(* IEC 61131-3 sources: HvIrBz/, 6 files *)

(* ---- d512.st ---- *)
if 取出物料盒1=1 THEN
	X轴绝对运动启动:=0;
	Z轴绝对运动启动:=0;
	X轴绝对运动位置设定 := 572;
    Z轴绝对运动位置设定 := 280;
	x回原点:=0;
	y回原点:=0;
	z回原点:=0;
(*	xz轴设定终了:=1;*)
	Y0 :=1;
	y3 :=0;
	Y1 :=0;
	X轴绝对运动速度设定:=50;
	Z轴绝对运动速度设定:=50;
	X轴绝对运动启动:=1;
	Z轴绝对运动启动:=1;

END_IF

if Z轴实时位置=280 and X轴实时位置=572 then
		旋转气缸:=1;
		Y轴绝对运动位置设定:=-188;
		Y轴绝对运动速度设定:=50;
		Y轴绝对运动启动:=1;
		y3 :=1;
END_IF

if 取出物料盒2=1 THEN
	X轴绝对运动位置设定 := 432;
    Z轴绝对运动位置设定 := 280;
x回原点:=0;
	y回原点:=0;
	z回原点:=0;
(*	xz轴设定终了:=1;*)
	Y0 :=1;
	y3 :=0;
	Y1 :=0;
	X轴绝对运动速度设定:=50;
	Z轴绝对运动速度设定:=50;
	X轴绝对运动启动:=1;
	Z轴绝对运动启动:=1;

END_IF

if Z轴实时位置=280 and X轴实时位置=432 then
		旋转气缸:=1;
		Y轴绝对运动位置设定:=-188;
		Y轴绝对运动速度设定:=50;
		Y轴绝对运动启动:=1;
		y3 :=1;
END_IF

if 取出物料盒3=1 THEN
	X轴绝对运动位置设定 := 292;
    Z轴绝对运动位置设定 := 280;
x回原点:=0;
	y回原点:=0;
	z回原点:=0;
(*	xz轴设定终了:=1;*)
	Y0 :=1;
	y3 :=0;
	Y1 :=0;
	X轴绝对运动速度设定:=50;
	Z轴绝对运动速度设定:=50;
	X轴绝对运动启动:=1;
	Z轴绝对运动启动:=1;

END_IF

if Z轴实时位置=280 and X轴实时位置=292 then
		旋转气缸:=1;
		Y轴绝对运动位置设定:=-188;
		Y轴绝对运动速度设定:=50;
		Y轴绝对运动启动:=1;
		y3 :=1;
		Y轴绝对运动启动:=0;
END_IF

if 取出物料盒4=1 THEN
	X轴绝对运动位置设定 := 152;
    Z轴绝对运动位置设定 := 280;
x回原点:=0;
	y回原点:=0;
	z回原点:=0;
(*	xz轴设定终了:=1;*)
	Y0 :=1;
	y3 :=0;
	Y1 :=0;
	X轴绝对运动速度设定:=50;
	Z轴绝对运动速度设定:=50;
	X轴绝对运动启动:=1;
	Z轴绝对运动启动:=1;
	X轴绝对运动启动:=0;
	Z轴绝对运动启动:=0;

END_IF

if Z轴实时位置=280 and X轴实时位置=152  then
		旋转气缸:=1;
		Z轴绝对运动启动:=0;
		Y轴绝对运动位置设定:=-188;
		Y轴绝对运动速度设定:=50;
		Y轴绝对运动启动:=1;
		Z轴绝对运动启动:=0;
		Y轴绝对运动启动:=0;
		y3 :=1;
END_IF

if 取出物料盒5=1 THEN
	X轴绝对运动位置设定 := 12;
    Z轴绝对运动位置设定 := 280;
x回原点:=0;
	y回原点:=0;
	z回原点:=0;
(*	xz轴设定终了:=1;*)
	Y0 :=1;
	y3 :=0;
	Y1 :=0;
	X轴绝对运动速度设定:=50;
	Z轴绝对运动速度设定:=50;
	X轴绝对运动启动:=1;
	Z轴绝对运动启动:=1;
	X轴绝对运动启动:=0;
	Z轴绝对运动启动:=0;

END_IF

if Z轴实时位置=280 and X轴实时位置=12  then
		旋转气缸:=1;
		Z轴绝对运动启动:=0;
		Y轴绝对运动位置设定:=-188;
		Y轴绝对运动速度设定:=50;
		Y轴绝对运动启动:=1;
		Z轴绝对运动启动:=0;
		Y轴绝对运动启动:=0;
		y3 :=1;
END_IF

(*if 取出物料盒6=1 THEN
	X轴绝对运动启动:=0;
	Z轴绝对运动启动:=0;
	X轴绝对运动位置设定 := 572;
    Z轴绝对运动位置设定 := 135;
x回原点:=0;
	y回原点:=0;
	z回原点:=0;
(*	xz轴设定终了:=1;*)
	Y0 :=1;
	y3 :=0;
	Y1 :=0;
	X轴绝对运动速度设定:=50;
	Z轴绝对运动速度设定:=50;
	X轴绝对运动启动:=1;
	Z轴绝对运动启动:=1;

END_IF

if Z轴实时位置=135 and X轴实时位置=572 and y3=0 then
		旋转气缸:=1;
		Y轴绝对运动位置设定:=-188;
		Y轴绝对运动速度设定:=50;
		Y轴绝对运动启动:=1;
		y3 :=1;
END_IF

if 取出物料盒7=1 THEN
	X轴绝对运动位置设定 := 432;
    Z轴绝对运动位置设定 := 135;
x回原点:=0;
	y回原点:=0;
	z回原点:=0;
(*	xz轴设定终了:=1;*)
	Y0 :=1;
	y3 :=0;
	Y1 :=0;
	X轴绝对运动速度设定:=50;
	Z轴绝对运动速度设定:=50;
	X轴绝对运动启动:=1;
	Z轴绝对运动启动:=1;

END_IF

if Z轴实时位置=135 and X轴实时位置=432 then
		旋转气缸:=1;
		Y轴绝对运动位置设定:=-188;
		Y轴绝对运动速度设定:=50;
		Y轴绝对运动启动:=1;
		y3 :=1;
END_IF

if 取出物料盒8=1 THEN
	X轴绝对运动位置设定 := 292;
    Z轴绝对运动位置设定 := 135;
x回原点:=0;
	y回原点:=0;
	z回原点:=0;
(*	xz轴设定终了:=1;*)
	Y0 :=1;
	y3 :=0;
	Y1 :=0;
	X轴绝对运动速度设定:=50;
	Z轴绝对运动速度设定:=50;
	X轴绝对运动启动:=1;
	Z轴绝对运动启动:=1;

END_IF

if Z轴实时位置=135 and X轴实时位置=292 then
		旋转气缸:=1;
		Y轴绝对运动位置设定:=-188;
		Y轴绝对运动速度设定:=50;
		Y轴绝对运动启动:=1;
		y3 :=1;
		Y轴绝对运动启动:=0;
END_IF

if 取出物料盒9=1 THEN
	X轴绝对运动位置设定 := 152;
    Z轴绝对运动位置设定 := 135;
x回原点:=0;
	y回原点:=0;
	z回原点:=0;
(*	xz轴设定终了:=1;*)
	Y0 :=1;
	y3 :=0;
	Y1 :=0;
	X轴绝对运动速度设定:=50;
	Z轴绝对运动速度设定:=50;
	X轴绝对运动启动:=1;
	Z轴绝对运动启动:=1;
	X轴绝对运动启动:=0;
	Z轴绝对运动启动:=0;

END_IF

if Z轴实时位置=135 and X轴实时位置=152 and 旋转气缸=0 then
		旋转气缸:=1;
		Z轴绝对运动启动:=0;
		Y轴绝对运动位置设定:=-188;
		Y轴绝对运动速度设定:=50;
		Y轴绝对运动启动:=1;
		Z轴绝对运动启动:=0;
		Y轴绝对运动启动:=0;
		y3 :=1;
END_IF

if 取出物料盒10=1 THEN
	X轴绝对运动位置设定 := 12;
    Z轴绝对运动位置设定 := 135;
x回原点:=0;
	y回原点:=0;
	z回原点:=0;
(*	xz轴设定终了:=1;*)
	Y0 :=1;
	y3 :=0;
	Y1 :=0;
	X轴绝对运动速度设定:=50;
	Z轴绝对运动速度设定:=50;
	X轴绝对运动启动:=1;
	Z轴绝对运动启动:=1;
	X轴绝对运动启动:=0;
	Z轴绝对运动启动:=0;

END_IF

if Z轴实时位置=135 and X轴实时位置=12 and 旋转气缸=0 then
		旋转气缸:=1;
		Z轴绝对运动启动:=0;
		Y轴绝对运动位置设定:=-188;
		Y轴绝对运动速度设定:=50;
		Y轴绝对运动启动:=1;
		Z轴绝对运动启动:=0;
		Y轴绝对运动启动:=0;
		y3 :=1;
END_IF

if 取出物料盒11=1 THEN
	X轴绝对运动启动:=0;
	Z轴绝对运动启动:=0;
	X轴绝对运动位置设定 := 572;
    Z轴绝对运动位置设定 := -10;
x回原点:=0;
	y回原点:=0;
	z回原点:=0;
(*	xz轴设定终了:=1;*)
	Y0 :=1;
	y3 :=0;
	Y1 :=0;
	X轴绝对运动速度设定:=50;
	Z轴绝对运动速度设定:=50;
	X轴绝对运动启动:=1;
	Z轴绝对运动启动:=1;

END_IF

if Z轴实时位置=-10 and X轴实时位置=572 and y3=0 then
		旋转气缸:=1;
		Y轴绝对运动位置设定:=-188;
		Y轴绝对运动速度设定:=50;
		Y轴绝对运动启动:=1;
		y3 :=1;
END_IF

if 取出物料盒12=1 THEN
	X轴绝对运动位置设定 := 432;
    Z轴绝对运动位置设定 := -10;
x回原点:=0;
	y回原点:=0;
	z回原点:=0;
(*	xz轴设定终了:=1;*)
	Y0 :=1;
	y3 :=0;
	Y1 :=0;
	X轴绝对运动速度设定:=50;
	Z轴绝对运动速度设定:=50;
	X轴绝对运动启动:=1;
	Z轴绝对运动启动:=1;

END_IF

if Z轴实时位置=-10 and X轴实时位置=432 then
		旋转气缸:=1;
		Y轴绝对运动位置设定:=-188;
		Y轴绝对运动速度设定:=50;
		Y轴绝对运动启动:=1;
		y3 :=1;
END_IF

if 取出物料盒13=1 THEN
	X轴绝对运动位置设定 := 292;
    Z轴绝对运动位置设定 := -10;
x回原点:=0;
	y回原点:=0;
	z回原点:=0;
(*	xz轴设定终了:=1;*)
	Y0 :=1;
	y3 :=0;
	Y1 :=0;
	X轴绝对运动速度设定:=50;
	Z轴绝对运动速度设定:=50;
	X轴绝对运动启动:=1;
	Z轴绝对运动启动:=1;

END_IF

if Z轴实时位置=-10 and X轴实时位置=292 then
		旋转气缸:=1;
		Y轴绝对运动位置设定:=-188;
		Y轴绝对运动速度设定:=50;
		Y轴绝对运动启动:=1;
		y3 :=1;
		Y轴绝对运动启动:=0;
END_IF

if 取出物料盒14=1 THEN
	X轴绝对运动位置设定 := 152;
    Z轴绝对运动位置设定 := -10;
x回原点:=0;
	y回原点:=0;
	z回原点:=0;
(*	xz轴设定终了:=1;*)
	Y0 :=1;
	y3 :=0;
	Y1 :=0;
	X轴绝对运动速度设定:=50;
	Z轴绝对运动速度设定:=50;
	X轴绝对运动启动:=1;
	Z轴绝对运动启动:=1;
	X轴绝对运动启动:=0;
	Z轴绝对运动启动:=0;

END_IF

if Z轴实时位置=-10 and X轴实时位置=152 and 旋转气缸=0 then
		旋转气缸:=1;
		Z轴绝对运动启动:=0;
		Y轴绝对运动位置设定:=-188;
		Y轴绝对运动速度设定:=50;
		Y轴绝对运动启动:=1;
		Z轴绝对运动启动:=0;
		Y轴绝对运动启动:=0;
		y3 :=1;
END_IF

if 取出物料盒15=1 THEN
	X轴绝对运动位置设定 := 12;
    Z轴绝对运动位置设定 := -10;
x回原点:=0;
	y回原点:=0;
	z回原点:=0;
(*	xz轴设定终了:=1;*)
	Y0 :=1;
	y3 :=0;
	Y1 :=0;
	X轴绝对运动速度设定:=50;
	Z轴绝对运动速度设定:=50;
	X轴绝对运动启动:=1;
	Z轴绝对运动启动:=1;
	X轴绝对运动启动:=0;
	Z轴绝对运动启动:=0;

END_IF

if Z轴实时位置=-10 and X轴实时位置=12 and 旋转气缸=0 then
		旋转气缸:=1;
		Z轴绝对运动启动:=0;
		Y轴绝对运动位置设定:=-188;
		Y轴绝对运动速度设定:=50;
		Y轴绝对运动启动:=1;
		Z轴绝对运动启动:=0;
		Y轴绝对运动启动:=0;
		y3 :=1;
END_IF*)

if x5=1 THEN
	Z轴绝对运动启动:=0;
	Y轴绝对运动启动:=0;
	END_IF

if Y轴实时位置=-188 then
	Z轴绝对运动启动:=0;
	Y轴绝对运动启动:=0;
	夹爪气缸:=1;
	y3:=0;
	Y2:=1;
	Z轴绝对运动位置设定:=285;
	Y轴绝对运动位置设定:=40;
	Z轴绝对运动速度设定:=50;
	Y轴绝对运动速度设定:=50;
(*	Z轴绝对运动启动:=1;
	Y轴绝对运动启动:=1;*)

	END_IF

if x6=1 THEN

	Z轴绝对运动启动:=1;
	Y轴绝对运动启动:=1;

	END_IF
(*if 取出物料盒2=1 or X6=1 THEN
	X轴绝对运动位置设定 := 432;
    Z轴绝对运动位置设定 := 280;

	xz轴设定终了:=1;
	Y1 :=1;
	Y0 :=0;
(*	X轴绝对运动启动:=1;
	Z轴绝对运动启动:=1;*)
END_IF

if 取出物料盒3=1 THEN
	X轴绝对运动位置设定 := 292;
    Z轴绝对运动位置设定 := 280;

	xz轴设定终了:=1;
	Y1 :=1;
	Y0 :=0;
(*	X轴绝对运动启动:=1;
	Z轴绝对运动启动:=1;*)
END_IF

if 取出物料盒4=1 THEN
	X轴绝对运动位置设定 := 152;
    Z轴绝对运动位置设定 := 280;

	xz轴设定终了:=1;
	Y1 :=1;
	Y0 :=0;
(*	X轴绝对运动启动:=1;
	Z轴绝对运动启动:=1;*)
END_IF

(*if 取出物料盒5=1 THEN
	X轴绝对运动位置设定 := 12;
    Z轴绝对运动位置设定 := 280;

	xz轴设定终了:=1;
	Y1 :=1;
	Y0 :=0;
	X轴绝对运动启动:=1;
	Z轴绝对运动启动:=1;
END_IF*)

if 取出物料盒1=1 or X6=1 THEN
	X轴绝对运动位置设定 := 432;
    Z轴绝对运动位置设定 := 280;

	xz轴设定终了:=1;
	Y1 :=1;
	Y0 :=0;
	X轴绝对运动启动:=1;
	Z轴绝对运动启动:=1;
END_IF

IF X5=1 THEN
	x回原点:=0;
	y回原点:=0;
	z回原点:=0;
	旋转气缸:=1;
	Y轴绝对运动位置设定:=-188;
	Y轴绝对运动速度设定:=50;
	X轴绝对运动速度设定:=50;
	Z轴绝对运动速度设定:=50;
	Y轴绝对运动启动:=1;
	X轴绝对运动启动:=1;
	Z轴绝对运动启动:=1;
	夹爪气缸:=1;
	IF Y轴实时位置=-188 THEN
	Y3:=1;
	END_IF;
END_IF*)

if X4=1 THEN
	旋转气缸:=0;
	x回原点:=1;
	y回原点:=1;
	z回原点:=1;
	X轴绝对运动启动:=0;
	Y轴绝对运动启动:=0;
	Z轴绝对运动启动:=0;
	END_IF

(* ---- d514.st ---- *)
if M8000=1 and 初始启动一次=0 THEN
	Z轴绝对运动启动:=0;
	X轴绝对运动启动:=0;
	Y轴绝对运动启动:=0;
	x回原点:=0;
	y回原点:=0;
	z回原点:=0;
	X轴绝对运动速度设定:=50;
	Z轴绝对运动速度设定:=50;
	y1:=1;
	d1301:=0;
	三轴启动:=0;
	初始启动一次:=1;
END_IF

IF 三轴启动=1 THEN
	X轴绝对运动速度设定:=50;
	Z轴绝对运动速度设定:=50;
	CASE 第一个运行 OF
		1:取出物料盒1:=1;
		2:取出物料盒2:=1;
		3:取出物料盒3:=1;
		4:取出物料盒4:=1;
		5:取出物料盒5:=1;
	Z轴绝对运动启动:=0;
	X轴绝对运动启动:=0;
	END_CASE;
END_IF;
if 取出物料盒1=1 and 取出物料盒只执行一次确保=0 THEN
	取出1:=1;
	X轴绝对运动位置设定 := 572;
    Z轴绝对运动位置设定 := 280;
	Z轴绝对运动启动:=1;
	取得是1:=1;
	取出物料盒只执行一次确保:=1;
END_IF
if 取出物料盒2=1 THEN
	取出1:=1;
	X轴绝对运动位置设定 := 432;
    Z轴绝对运动位置设定 := 280;
	Z轴绝对运动启动:=1;
	取得是2:=1;

END_IF
if  取出物料盒3=1  THEN
	取出1:=1;
	X轴绝对运动位置设定 := 292;
    Z轴绝对运动位置设定 := 280;
	Z轴绝对运动启动:=1;
	取得是3:=1;
END_IF
if 取出物料盒4=1 THEN
	取出1:=1;
	X轴绝对运动位置设定 := 152;
    Z轴绝对运动位置设定 := 280;
	Z轴绝对运动启动:=1;
	取得是4:=1;
END_IF
if  取出物料盒5=1 THEN
	取出1:=1;
	X轴绝对运动位置设定 := 12;
    Z轴绝对运动位置设定 := 280;
	Z轴绝对运动启动:=1;
	取得是5:=1;
END_IF
	IF Z轴实时位置>20 and 取得是1=1  THEN

		X轴绝对运动启动:=1;
	END_IF;

	IF Z轴实时位置>20 and 取得是2=1  THEN

		X轴绝对运动启动:=1;
	END_IF;

	IF Z轴实时位置>20 and 取得是3=1  THEN

		X轴绝对运动启动:=1;
	END_IF;

	IF Z轴实时位置>20 and 取得是4=1  THEN

		X轴绝对运动启动:=1;
	END_IF;

	IF Z轴实时位置>20 and 取得是5=1  THEN

		X轴绝对运动启动:=1;
	END_IF;
if Z轴实时位置=280 and X轴实时位置=572 and 取得是1=1 then
		旋转气缸:=1;
		Y轴绝对运动位置设定:=-188;
		Y轴绝对运动速度设定:=50;
		Y轴绝对运动启动:=1;
		y3 :=1;
		Z轴绝对运动启动:=0;
END_IF

if Z轴实时位置=280 and X轴实时位置=432 and 取得是2=1 then
		旋转气缸:=1;
		Y轴绝对运动位置设定:=-188;
		Y轴绝对运动速度设定:=50;
		Y轴绝对运动启动:=1;
		y3 :=1;
END_IF

if Z轴实时位置=280 and X轴实时位置=292 and 取得是3=1 then
		旋转气缸:=1;
		Y轴绝对运动位置设定:=-188;
		Y轴绝对运动速度设定:=50;
		Y轴绝对运动启动:=1;
		y3 :=1;
END_IF

if Z轴实时位置=280 and X轴实时位置=152 and 取得是4=1 then
		旋转气缸:=1;
		Y轴绝对运动位置设定:=-188;
		Y轴绝对运动速度设定:=50;
		Y轴绝对运动启动:=1;
		y3 :=1;
END_IF
if Z轴实时位置=280 and X轴实时位置=12 and 取得是5=1 then
		旋转气缸:=1;
		Y轴绝对运动位置设定:=-188;
		Y轴绝对运动速度设定:=50;
		Y轴绝对运动启动:=1;
		y3 :=1;
END_IF
if Y轴实时位置=-188 then
	Z轴绝对运动启动:=0;
	Y轴绝对运动启动:=0;
	夹爪气缸:=1;
	y3:=0;
	Y2:=1;
	Z轴绝对运动位置设定:=285;
	Y轴绝对运动位置设定:=40;
	Z轴绝对运动速度设定:=50;
	Y轴绝对运动速度设定:=50;
	X轴绝对运动位置设定:=303;
	Z轴绝对运动启动:=1;
	END_IF

IF Z轴实时位置=285 THEN

	Y轴绝对运动启动:=1;
	运动状态:=0;
	取料终:=1;
END_IF;

(*IF x5=1 THEN
	Z轴绝对运动启动:=1;
	Y轴绝对运动启动:=1;
	运动状态:=0;
	取料终:=1;
END_IF;*)

IF 取料终=1 and Y轴实时位置>35 THEN
	旋转气缸:=0;
	X轴绝对运动启动:=1;
	放到顶上了:=1;
	Z轴绝对运动启动:=0;
	Y轴绝对运动启动:=0;
	Y2:=1;
END_IF;

IF 放到顶上了=1 and X轴实时位置=303 THEN
	Z轴绝对运动位置设定:=0;
	Z轴绝对运动启动:=1;
	Y轴绝对运动启动:=1;
	X轴绝对运动启动:=1;
	Y3:=1;
	放完了:=1;
END_IF;

IF 放完了=1 and Z轴实时位置=0 THEN
	夹爪气缸:=0;
	x回原点:=1;
	y回原点:=1;
	z回原点:=1;
END_IF;

(* ---- d515.st ---- *)
if M8000=1 and 初始启动一次=0 THEN
	Z轴绝对运动启动:=0;
	X轴绝对运动启动:=0;
	Y轴绝对运动启动:=0;
	x回原点:=0;
	y回原点:=0;
	z回原点:=0;
	X轴绝对运动速度设定:=50;
	Z轴绝对运动速度设定:=50;

	d1301:=0;
	三轴启动:=0;
	圆形落料:=0;
	初始启动一次:=1;

END_IF

IF 三轴启动=1 THEN
	传送带速度:=50;
	传送带位置:=20000;
	圆形物料推料气缸:=1;

	切换吸盘:=1;

	X轴绝对运动速度设定:=50;
	Z轴绝对运动速度设定:=50;
	CASE 第一个运行 OF
		1:取出物料盒1:=1;
		2:取出物料盒2:=1;
		3:取出物料盒3:=1;
		4:取出物料盒4:=1;
		5:取出物料盒5:=1;
		6:取出物料盒6:=1;
		7:取出物料盒7:=1;
		8:取出物料盒8:=1;
		9:取出物料盒9:=1;
		10:取出物料盒10:=1;
		11:取出物料盒11:=1;
		12:取出物料盒12:=1;
		13:取出物料盒13:=1;
		14:取出物料盒14:=1;
		15:取出物料盒15:=1;

	Z轴绝对运动启动:=0;
	X轴绝对运动启动:=0;
	END_CASE;
END_IF;
if 取出物料盒1=1 and 取出物料盒只执行一次确保=0 THEN
	取出1:=1;
	X轴绝对运动位置设定 := 572;
    Z轴绝对运动位置设定 := 280;
	Z轴绝对运动启动:=1;
	取得是1:=1;
	取出物料盒只执行一次确保:=1;
END_IF
if 取出物料盒2=1 and 取出物料盒只执行一次确保=0 THEN
	取出1:=1;
	X轴绝对运动位置设定 := 432;
    Z轴绝对运动位置设定 := 280;
	Z轴绝对运动启动:=1;
	取得是2:=1;
	取出物料盒只执行一次确保:=1;
END_IF
if  取出物料盒3=1 and 取出物料盒只执行一次确保=0  THEN
	取出1:=1;
	X轴绝对运动位置设定 := 292;
    Z轴绝对运动位置设定 := 280;
	Z轴绝对运动启动:=1;
	取得是3:=1;
	取出物料盒只执行一次确保:=1;
END_IF
if 取出物料盒4=1 and 取出物料盒只执行一次确保=0 THEN
	取出1:=1;
	X轴绝对运动位置设定 := 152;
    Z轴绝对运动位置设定 := 280;
	Z轴绝对运动启动:=1;
	取得是4:=1;
	取出物料盒只执行一次确保:=1;
END_IF
if  取出物料盒5=1 and 取出物料盒只执行一次确保=0 THEN
	取出1:=1;
	X轴绝对运动位置设定 := 12;
    Z轴绝对运动位置设定 := 280;
	Z轴绝对运动启动:=1;
	取得是5:=1;
	取出物料盒只执行一次确保:=1;
END_IF
if 取出物料盒6=1 and 取出物料盒只执行一次确保=0 THEN
	取出1:=1;
	X轴绝对运动位置设定 := 572;
    Z轴绝对运动位置设定 := 135;
	Z轴绝对运动启动:=1;
	取得是6:=1;
	取出物料盒只执行一次确保:=1;

END_IF
if 取出物料盒7=1 and 取出物料盒只执行一次确保=0 THEN
	取出1:=1;
	X轴绝对运动位置设定 := 432;
    Z轴绝对运动位置设定 := 135;
	Z轴绝对运动启动:=1;
	取得是7:=1;
	取出物料盒只执行一次确保:=1;
END_IF
if  取出物料盒8=1 and 取出物料盒只执行一次确保=0  THEN
	取出1:=1;
	X轴绝对运动位置设定 := 292;
    Z轴绝对运动位置设定 := 135;
	Z轴绝对运动启动:=1;
	取得是8:=1;
	取出物料盒只执行一次确保:=1;
END_IF
if 取出物料盒9=1 and 取出物料盒只执行一次确保=0 THEN
	取出1:=1;
	X轴绝对运动位置设定 := 152;
    Z轴绝对运动位置设定 := 135;
	Z轴绝对运动启动:=1;
	取得是9:=1;
	取出物料盒只执行一次确保:=1;
END_IF
if  取出物料盒10=1 and 取出物料盒只执行一次确保=0 THEN
	取出1:=1;
	X轴绝对运动位置设定 := 12;
    Z轴绝对运动位置设定 := 135;
	Z轴绝对运动启动:=1;
	取得是10:=1;
	取出物料盒只执行一次确保:=1;
END_IF
if 取出物料盒11=1 and 取出物料盒只执行一次确保=0 THEN
	取出1:=1;
	X轴绝对运动位置设定 := 572;
    Z轴绝对运动位置设定 := -10;
	Z轴绝对运动启动:=1;
	取得是11:=1;
	取出物料盒只执行一次确保:=1;
END_IF
if 取出物料盒12=1 and 取出物料盒只执行一次确保=0 THEN
	取出1:=1;
	X轴绝对运动位置设定 := 432;
    Z轴绝对运动位置设定 := -10;
	Z轴绝对运动启动:=1;
	取得是12:=1;
	取出物料盒只执行一次确保:=1;
END_IF
if  取出物料盒13=1 and 取出物料盒只执行一次确保=0  THEN
	取出1:=1;
	X轴绝对运动位置设定 := 292;
    Z轴绝对运动位置设定 := -10;
	Z轴绝对运动启动:=1;
	取得是13:=1;
	取出物料盒只执行一次确保:=1;
END_IF
if 取出物料盒14=1 and 取出物料盒只执行一次确保=0 THEN
	取出1:=1;
	X轴绝对运动位置设定 := 152;
    Z轴绝对运动位置设定 := -10;
	Z轴绝对运动启动:=1;
	取得是14:=1;
	取出物料盒只执行一次确保:=1;
END_IF
if  取出物料盒15=1 and 取出物料盒只执行一次确保=0 THEN
	取出1:=1;
	X轴绝对运动位置设定 := 12;
    Z轴绝对运动位置设定 := -10;
	Z轴绝对运动启动:=1;
	取得是15:=1;
	取出物料盒只执行一次确保:=1;
END_IF
	IF Z轴实时位置>20 and 取得是1=1 and 确保x轴只动一次=0 THEN
		确保x轴只动一次:=1;
		X轴绝对运动启动:=1;
	END_IF;
	IF Z轴实时位置>20 and 取得是2=1 and 确保x轴只动一次=0  THEN
		确保x轴只动一次:=1;
		X轴绝对运动启动:=1;
		传送带启动:=1;
	END_IF;

	IF Z轴实时位置>20 and 取得是3=1 and 确保x轴只动一次=0  THEN
		确保x轴只动一次:=1;
		X轴绝对运动启动:=1;
	END_IF;

	IF Z轴实时位置>20 and 取得是4=1 and 确保x轴只动一次=0  THEN
		确保x轴只动一次:=1;
		X轴绝对运动启动:=1;
	END_IF;

	IF Z轴实时位置>20 and 取得是5=1 and 确保x轴只动一次=0  THEN
		确保x轴只动一次:=1;
		X轴绝对运动启动:=1;
	END_IF;
	IF Z轴实时位置>20 and 取得是6=1 and 确保x轴只动一次=0 THEN
		确保x轴只动一次:=1;

		X轴绝对运动启动:=1;
		传送带启动:=1;
	END_IF;
	IF Z轴实时位置>20 and 取得是7=1 and 确保x轴只动一次=0  THEN
		确保x轴只动一次:=1;
		X轴绝对运动启动:=1;
		传送带启动:=1;
	END_IF;

	IF Z轴实时位置>20 and 取得是8=1 and 确保x轴只动一次=0  THEN
		确保x轴只动一次:=1;
		X轴绝对运动启动:=1;
	END_IF;

	IF Z轴实时位置>20 and 取得是9=1 and 确保x轴只动一次=0  THEN
		确保x轴只动一次:=1;
		X轴绝对运动启动:=1;
	END_IF;

	IF Z轴实时位置>20 and 取得是10=1 and 确保x轴只动一次=0  THEN
		确保x轴只动一次:=1;
		X轴绝对运动启动:=1;
	END_IF;
	IF Z轴实时位置<-2 and 取得是11=1 and 确保x轴只动一次=0 THEN
		确保x轴只动一次:=1;
		X轴绝对运动启动:=1;
	END_IF;
	IF Z轴实时位置<-2 and 取得是12=1 and 确保x轴只动一次=0  THEN
		确保x轴只动一次:=1;
		X轴绝对运动启动:=1;
		传送带启动:=1;
	END_IF;

	IF Z轴实时位置<-2 and 取得是13=1 and 确保x轴只动一次=0  THEN
		确保x轴只动一次:=1;
		X轴绝对运动启动:=1;
	END_IF;

	IF Z轴实时位置<-2 and 取得是14=1 and 确保x轴只动一次=0  THEN
		确保x轴只动一次:=1;
		X轴绝对运动启动:=1;
	END_IF;

	IF Z轴实时位置<-2 and 取得是15=1 and 确保x轴只动一次=0  THEN
		确保x轴只动一次:=1;
		X轴绝对运动启动:=1;
	END_IF;
IF Z轴实时位置>30 and 第一个=0 THEN
	圆形物料推料气缸:=0;
	一号物料完工:=1;
	END_IF
if Z轴实时位置=280 and X轴实时位置=572 and 取得是1=1 then
		旋转气缸:=1;
		Y轴绝对运动位置设定:=-188;
		Y轴绝对运动速度设定:=50;
		Y轴绝对运动启动:=1;
		y3 :=1;
		Z轴绝对运动启动:=0;
END_IF

if Z轴实时位置=280 and X轴实时位置=432 and 取得是2=1 then
		旋转气缸:=1;
		Y轴绝对运动位置设定:=-188;
		Y轴绝对运动速度设定:=50;
		Y轴绝对运动启动:=1;
		y3 :=1;
END_IF

if Z轴实时位置=280 and X轴实时位置=292 and 取得是3=1 then
		旋转气缸:=1;
		Y轴绝对运动位置设定:=-188;
		Y轴绝对运动速度设定:=50;
		Y轴绝对运动启动:=1;
		y3 :=1;
END_IF

if Z轴实时位置=280 and X轴实时位置=152 and 取得是4=1 then
		旋转气缸:=1;
		Y轴绝对运动位置设定:=-188;
		Y轴绝对运动速度设定:=50;
		Y轴绝对运动启动:=1;
		y3 :=1;
END_IF
if Z轴实时位置=280 and X轴实时位置=12 and 取得是5=1 then
		旋转气缸:=1;
		Y轴绝对运动位置设定:=-188;
		Y轴绝对运动速度设定:=50;
		Y轴绝对运动启动:=1;
		y3 :=1;
END_IF
if Z轴实时位置=135 and X轴实时位置=572 and 取得是6=1 then
		旋转气缸:=1;
		Y轴绝对运动位置设定:=-188;
		Y轴绝对运动速度设定:=50;
		Y轴绝对运动启动:=1;

		Z轴绝对运动启动:=0;

			第一个:=1;
END_IF

if Z轴实时位置=135 and X轴实时位置=432 and 取得是7=1 then
		旋转气缸:=1;
		Y轴绝对运动位置设定:=-188;
		Y轴绝对运动速度设定:=50;
		Y轴绝对运动启动:=1;
		y3 :=1;
END_IF

if Z轴实时位置=135 and X轴实时位置=292 and 取得是8=1 then
		旋转气缸:=1;
		Y轴绝对运动位置设定:=-188;
		Y轴绝对运动启动:=1;
		y3 :=1;
END_IF

if Z轴实时位置=135 and X轴实时位置=152 and 取得是9=1 then
		旋转气缸:=1;
		Y轴绝对运动位置设定:=-188;
		Y轴绝对运动速度设定:=50;
		Y轴绝对运动启动:=1;
		y3 :=1;
END_IF
if Z轴实时位置=135 and X轴实时位置=12 and 取得是10=1 then
		旋转气缸:=1;
		Y轴绝对运动位置设定:=-188;
		Y轴绝对运动速度设定:=50;
		Y轴绝对运动启动:=1;
		y3 :=1;
END_IF
if X轴实时位置=572 and 取得是11=1 then
		旋转气缸:=1;
		Y轴绝对运动位置设定:=-188;
		Y轴绝对运动速度设定:=50;
		Y轴绝对运动启动:=1;
		y3 :=1;
		Z轴绝对运动启动:=0;
END_IF

if X轴实时位置=432 and 取得是12=1 then
		旋转气缸:=1;
		Y轴绝对运动位置设定:=-188;
		Y轴绝对运动速度设定:=50;
		Y轴绝对运动启动:=1;
		y3 :=1;
END_IF

if X轴实时位置=292 and 取得是13=1 then
		旋转气缸:=1;
		Y轴绝对运动位置设定:=-188;
		Y轴绝对运动速度设定:=50;
		Y轴绝对运动启动:=1;
		y3 :=1;
END_IF

if X轴实时位置=152 and 取得是14=1 then
		旋转气缸:=1;
		Y轴绝对运动位置设定:=-188;
		Y轴绝对运动速度设定:=50;
		Y轴绝对运动启动:=1;
		y3 :=1;
END_IF
if X轴实时位置=12 and 取得是15=1 then
		旋转气缸:=1;
		Y轴绝对运动位置设定:=-188;
		Y轴绝对运动速度设定:=50;
		Y轴绝对运动启动:=1;
		y3 :=1;
END_IF
if Y轴实时位置=-188 and Z轴实时位置<0 then
	X轴绝对运动启动:=0;
	Z轴绝对运动启动:=0;
	Y轴绝对运动启动:=0;
	夹爪气缸:=1;
	y3:=0;
	Y2:=1;

	Z轴绝对运动位置设定:=-5;
	Y轴绝对运动位置设定:=40;
	Z轴绝对运动速度设定:=40;
	Y轴绝对运动速度设定:=50;
	X轴绝对运动位置设定:=303;

	夹爪完了:=1;
END_IF
if Y轴实时位置=-188 and Z轴实时位置=280 then
	X轴绝对运动启动:=0;
	Z轴绝对运动启动:=0;
	Y轴绝对运动启动:=0;
	夹爪气缸:=1;
	y3:=0;
	Y2:=1;

	Z轴绝对运动位置设定:=285;
	Y轴绝对运动位置设定:=40;
	Z轴绝对运动速度设定:=40;
	Y轴绝对运动速度设定:=50;
	X轴绝对运动位置设定:=303;

	夹爪完了:=1;
END_IF
if Y轴实时位置=-188 and Z轴实时位置=135 then
	X轴绝对运动启动:=0;
	Z轴绝对运动启动:=0;
	Y轴绝对运动启动:=0;
	夹爪气缸:=1;
	y3:=0;
	Y2:=1;

	Z轴绝对运动位置设定:=140;
	Y轴绝对运动位置设定:=40;
	Z轴绝对运动速度设定:=40;
	Y轴绝对运动速度设定:=50;
	X轴绝对运动位置设定:=303;

	夹爪完了:=1;
END_IF
TONR(IN := 夹爪完了,PT := 1000,Q => 开始带走);
TONR(IN := 夹爪完了,PT := 1200,Q => 开始带走2);
IF 开始带走=1 THEN
	Z轴绝对运动启动:=1;

	运动状态:=0;
	取料终:=1;
END_IF;
if 开始带走2=1 THEN
	Y轴绝对运动启动:=1;
END_if

IF 取料终=1 and Y轴实时位置>35 THEN
	旋转气缸:=0;
	X轴绝对运动启动:=1;
	放到顶上了:=1;
	Z轴绝对运动启动:=0;
	Y轴绝对运动启动:=0;
	Y2:=1;
END_IF;

IF 放到顶上了=1 and X轴实时位置=303 THEN
	Z轴绝对运动位置设定:=0;
	Z轴绝对运动启动:=1;
	Y轴绝对运动启动:=1;
	X轴绝对运动启动:=1;
	Y3:=1;
	放完了:=1;
END_IF;
TONR(IN := 放完了,PT := 200,Q => 真放完了);
IF 真放完了=1 THEN
	Z轴绝对运动启动:=0;
END_IF;
IF 放完了=1 and Z轴实时位置=0 THEN

	夹爪气缸:=0;
	最后放完了:=1;
	绝对放完了:=1;

END_IF;
TONR(IN := 最后放完了,PT := 200,Q => 最后放完了延时);

IF 最后放完了延时=1 THEN
	Z轴绝对运动位置设定:=40;
	Z轴绝对运动启动:=1;
	绝对放完了:=1;
END_IF;
IF Z轴实时位置>39 and 绝对放完了=1 THEN
	x回原点:=1;
	(*y回原点:=1;*)
	z回原点:=1;
	旋转气缸:=0;

	方形物料推料气缸:=1;
END_IF;
IF 一号传感器=1 THEN
	六轴机器人启动:=0;
END_IF;
if 二号传感器=1 THEN
	六轴机器人动作预备:=1;
END_IF

TONR(IN := 六轴机器人动作预备,PT := 7000,Q => 六轴机器人动作);

IF 六轴机器人动作=1 and 放完了=1 THEN
	六轴机器人启动:=1;
	六轴机器人动作预备:=0;

END_IF;
if 六轴作业完成=1 and 二号物料完工=0 and 绝对放完了=1 THEN
	二号物料完工:=1;
	方形物料推料气缸:=0;
	END_IF
TONR(IN := 二号物料完工,PT := 25000,Q => 三号物料完工);

IF 三号物料完工=1 THEN

	方形物料推料气缸:=0;
END_IF;
IF X4=1 THEN
	圆形物料推料气缸:=0;
END_IF;
IF X5=1 THEN
	方形物料推料气缸:=0;
END_IF;

(* ---- d516.st ---- *)
if M8000=1 and 初始启动一次=0 and x2=1 THEN
	Z轴绝对运动启动:=0;
	X轴绝对运动启动:=0;
	Y轴绝对运动启动:=0;
	x回原点:=0;
	y回原点:=0;
	z回原点:=0;
	X轴绝对运动速度设定:=50;
	Z轴绝对运动速度设定:=50;

	d1301:=0;
	三轴启动:=0;
	圆形落料:=0;
	初始启动一次:=1;

END_IF

IF (三轴启动=1 or x0=1)  and x2=1 THEN
	传送带速度:=50;
	传送带位置:=20000;
	圆形物料推料气缸:=1;

	切换吸盘:=1;

	X轴绝对运动速度设定:=50;
	Z轴绝对运动速度设定:=50;
	CASE 第一个运行 OF
		1:取出物料盒1:=1;
		2:取出物料盒2:=1;
		3:取出物料盒3:=1;
		4:取出物料盒4:=1;
		5:取出物料盒5:=1;
		6:取出物料盒6:=1;
		7:取出物料盒7:=1;
		8:取出物料盒8:=1;
		9:取出物料盒9:=1;
		10:取出物料盒10:=1;
		11:取出物料盒11:=1;
		12:取出物料盒12:=1;
		13:取出物料盒13:=1;
		14:取出物料盒14:=1;
		15:取出物料盒15:=1;

	Z轴绝对运动启动:=0;
	X轴绝对运动启动:=0;
	END_CASE;
END_IF;
if 取出物料盒1=1 and 取出物料盒只执行一次确保=0 and x2=1 THEN
	取出1:=1;
	X轴绝对运动位置设定 := 572;
    Z轴绝对运动位置设定 := 280;
	Z轴绝对运动启动:=1;
	取得是1:=1;
	取出物料盒只执行一次确保:=1;
END_IF
if 取出物料盒2=1 and 取出物料盒只执行一次确保=0 and x2=1 THEN
	取出1:=1;
	X轴绝对运动位置设定 := 432;
    Z轴绝对运动位置设定 := 280;
	Z轴绝对运动启动:=1;
	取得是2:=1;
	取出物料盒只执行一次确保:=1;
END_IF
if  取出物料盒3=1 and 取出物料盒只执行一次确保=0 and x2=1  THEN
	取出1:=1;
	X轴绝对运动位置设定 := 292;
    Z轴绝对运动位置设定 := 280;
	Z轴绝对运动启动:=1;
	取得是3:=1;
	取出物料盒只执行一次确保:=1;
END_IF
if 取出物料盒4=1 and 取出物料盒只执行一次确保=0 and x2=1 THEN
	取出1:=1;
	X轴绝对运动位置设定 := 152;
    Z轴绝对运动位置设定 := 280;
	Z轴绝对运动启动:=1;
	取得是4:=1;
	取出物料盒只执行一次确保:=1;
END_IF
if  取出物料盒5=1 and 取出物料盒只执行一次确保=0 and x2=1 THEN
	取出1:=1;
	X轴绝对运动位置设定 := 12;
    Z轴绝对运动位置设定 := 280;
	Z轴绝对运动启动:=1;
	取得是5:=1;
	取出物料盒只执行一次确保:=1;
END_IF
if 取出物料盒6=1 and 取出物料盒只执行一次确保=0 and x2=1 THEN
	取出1:=1;
	X轴绝对运动位置设定 := 572;
    Z轴绝对运动位置设定 := 135;
	Z轴绝对运动启动:=1;
	取得是6:=1;
	取出物料盒只执行一次确保:=1;

END_IF
if 取出物料盒7=1 and 取出物料盒只执行一次确保=0  and x2=1 THEN
	取出1:=1;
	X轴绝对运动位置设定 := 432;
    Z轴绝对运动位置设定 := 135;
	Z轴绝对运动启动:=1;
	取得是7:=1;
	取出物料盒只执行一次确保:=1;
END_IF
if  取出物料盒8=1 and 取出物料盒只执行一次确保=0  and x2=1 THEN
	取出1:=1;
	X轴绝对运动位置设定 := 292;
    Z轴绝对运动位置设定 := 135;
	Z轴绝对运动启动:=1;
	取得是8:=1;
	取出物料盒只执行一次确保:=1;
END_IF
if 取出物料盒9=1 and 取出物料盒只执行一次确保=0 and x2=1 THEN
	取出1:=1;
	X轴绝对运动位置设定 := 152;
    Z轴绝对运动位置设定 := 135;
	Z轴绝对运动启动:=1;
	取得是9:=1;
	取出物料盒只执行一次确保:=1;
END_IF
if  取出物料盒10=1 and 取出物料盒只执行一次确保=0 and x2=1 THEN
	取出1:=1;
	X轴绝对运动位置设定 := 12;
    Z轴绝对运动位置设定 := 135;
	Z轴绝对运动启动:=1;
	取得是10:=1;
	取出物料盒只执行一次确保:=1;
END_IF
if 取出物料盒11=1 and 取出物料盒只执行一次确保=0 and x2=1 THEN
	取出1:=1;
	X轴绝对运动位置设定 := 572;
    Z轴绝对运动位置设定 := -10;
	Z轴绝对运动启动:=1;
	取得是11:=1;
	取出物料盒只执行一次确保:=1;
END_IF
if 取出物料盒12=1 and 取出物料盒只执行一次确保=0 and x2=1 THEN
	取出1:=1;
	X轴绝对运动位置设定 := 432;
    Z轴绝对运动位置设定 := -10;
	Z轴绝对运动启动:=1;
	取得是12:=1;
	取出物料盒只执行一次确保:=1;
END_IF
if  取出物料盒13=1 and 取出物料盒只执行一次确保=0  and x2=1 THEN
	取出1:=1;
	X轴绝对运动位置设定 := 292;
    Z轴绝对运动位置设定 := -10;
	Z轴绝对运动启动:=1;
	取得是13:=1;
	取出物料盒只执行一次确保:=1;
END_IF
if 取出物料盒14=1 and 取出物料盒只执行一次确保=0 and x2=1 THEN
	取出1:=1;
	X轴绝对运动位置设定 := 152;
    Z轴绝对运动位置设定 := -10;
	Z轴绝对运动启动:=1;
	取得是14:=1;
	取出物料盒只执行一次确保:=1;
END_IF
if  取出物料盒15=1 and 取出物料盒只执行一次确保=0  and x2=1 THEN
	取出1:=1;
	X轴绝对运动位置设定 := 12;
    Z轴绝对运动位置设定 := -10;
	Z轴绝对运动启动:=1;
	取得是15:=1;
	取出物料盒只执行一次确保:=1;
END_IF
	IF Z轴实时位置>20 and 取得是1=1 and 确保x轴只动一次=0 and 回收作业启动=0 and x2=1 THEN
		确保x轴只动一次:=1;
		X轴绝对运动启动:=1;
	END_IF;
	IF Z轴实时位置>20 and 取得是2=1 and 确保x轴只动一次=0 and 回收作业启动=0 and x2=1  THEN
		确保x轴只动一次:=1;
		X轴绝对运动启动:=1;
		传送带启动:=1;
	END_IF;

	IF Z轴实时位置>20 and 取得是3=1 and 确保x轴只动一次=0 and 回收作业启动=0 and x2=1  THEN
		确保x轴只动一次:=1;
		X轴绝对运动启动:=1;
	END_IF;

	IF Z轴实时位置>20 and 取得是4=1 and 确保x轴只动一次=0 and 回收作业启动=0  and x2=1 THEN
		确保x轴只动一次:=1;
		X轴绝对运动启动:=1;
	END_IF;

	IF Z轴实时位置>20 and 取得是5=1 and 确保x轴只动一次=0 and 回收作业启动=0  and x2=1 THEN
		确保x轴只动一次:=1;
		X轴绝对运动启动:=1;
	END_IF;
	IF Z轴实时位置>20 and 取得是6=1 and 确保x轴只动一次=0 and 回收作业启动=0 and x2=1 THEN
		确保x轴只动一次:=1;

		X轴绝对运动启动:=1;
		传送带启动:=1;
	END_IF;
	IF Z轴实时位置>20 and 取得是7=1 and 确保x轴只动一次=0 and 回收作业启动=0 and x2=1  THEN
		确保x轴只动一次:=1;
		X轴绝对运动启动:=1;
		传送带启动:=1;
	END_IF;

	IF Z轴实时位置>20 and 取得是8=1 and 确保x轴只动一次=0 and 回收作业启动=0 and x2=1  THEN
		确保x轴只动一次:=1;
		X轴绝对运动启动:=1;
	END_IF;

	IF Z轴实时位置>20 and 取得是9=1 and 确保x轴只动一次=0 and 回收作业启动=0 and x2=1  THEN
		确保x轴只动一次:=1;
		X轴绝对运动启动:=1;
	END_IF;

	IF Z轴实时位置>20 and 取得是10=1 and 确保x轴只动一次=0 and 回收作业启动=0 and x2=1  THEN
		确保x轴只动一次:=1;
		X轴绝对运动启动:=1;
	END_IF;
	IF Z轴实时位置<-2 and 取得是11=1 and 确保x轴只动一次=0 and 回收作业启动=0 and x2=1 THEN
		确保x轴只动一次:=1;
		X轴绝对运动启动:=1;
	END_IF;
	IF Z轴实时位置<-2 and 取得是12=1 and 确保x轴只动一次=0 and 回收作业启动=0  and x2=1 THEN
		确保x轴只动一次:=1;
		X轴绝对运动启动:=1;
		传送带启动:=1;
	END_IF;

	IF Z轴实时位置<-2 and 取得是13=1 and 确保x轴只动一次=0  and 回收作业启动=0 and x2=1 THEN
		确保x轴只动一次:=1;
		X轴绝对运动启动:=1;
	END_IF;

	IF Z轴实时位置<-2 and 取得是14=1 and 确保x轴只动一次=0  and 回收作业启动=0 and x2=1 THEN
		确保x轴只动一次:=1;
		X轴绝对运动启动:=1;
	END_IF;

	IF Z轴实时位置<-2 and 取得是15=1 and 确保x轴只动一次=0 and 回收作业启动=0 and x2=1  THEN
		确保x轴只动一次:=1;
		X轴绝对运动启动:=1;
	END_IF;
IF Z轴实时位置>30 and 第一个=0 and 回收作业启动=0 and x2=1 THEN
	圆形物料推料气缸:=0;
	一号物料完工:=1;
	END_IF
if Z轴实时位置=280 and X轴实时位置=572 and 取得是1=1 and x2=1 then
		旋转气缸:=1;
		Y轴绝对运动位置设定:=-188;
		Y轴绝对运动速度设定:=50;
		Y轴绝对运动启动:=1;
		Z轴绝对运动启动:=0;
		第一个:=1;
END_IF

if Z轴实时位置=280 and X轴实时位置=432 and 取得是2=1 and x2=1 then
		旋转气缸:=1;
		Y轴绝对运动位置设定:=-188;
		Y轴绝对运动速度设定:=50;
		Y轴绝对运动启动:=1;
		Z轴绝对运动启动:=0;
		第一个:=1;
END_IF

if Z轴实时位置=280 and X轴实时位置=292 and 取得是3=1 and x2=1 then
		旋转气缸:=1;
		Y轴绝对运动位置设定:=-188;
		Y轴绝对运动速度设定:=50;
		Y轴绝对运动启动:=1;
		Z轴绝对运动启动:=0;
		第一个:=1;
END_IF

if Z轴实时位置=280 and X轴实时位置=152 and 取得是4=1 and x2=1 then
		旋转气缸:=1;
		Y轴绝对运动位置设定:=-188;
		Y轴绝对运动速度设定:=50;
		Y轴绝对运动启动:=1;
		Z轴绝对运动启动:=0;
		第一个:=1;
END_IF
if Z轴实时位置=280 and X轴实时位置=12 and 取得是5=1 and x2=1 then
		旋转气缸:=1;
		Y轴绝对运动位置设定:=-188;
		Y轴绝对运动速度设定:=50;
		Y轴绝对运动启动:=1;
		Z轴绝对运动启动:=0;
		第一个:=1;
END_IF
if Z轴实时位置=135 and X轴实时位置=572 and 取得是6=1 and x2=1 then
		旋转气缸:=1;
		Y轴绝对运动位置设定:=-188;
		Y轴绝对运动速度设定:=50;
		Y轴绝对运动启动:=1;

		Z轴绝对运动启动:=0;
		第一个:=1;
END_IF

if Z轴实时位置=135 and X轴实时位置=432 and 取得是7=1 and x2=1 then
		旋转气缸:=1;
		Y轴绝对运动位置设定:=-188;
		Y轴绝对运动速度设定:=50;
		Y轴绝对运动启动:=1;
		Z轴绝对运动启动:=0;
		第一个:=1;
END_IF

if Z轴实时位置=135 and X轴实时位置=292 and 取得是8=1 and x2=1 then
		旋转气缸:=1;
		Y轴绝对运动位置设定:=-188;
		Y轴绝对运动启动:=1;
		Z轴绝对运动启动:=0;
		第一个:=1;
END_IF

if Z轴实时位置=135 and X轴实时位置=152 and 取得是9=1 and x2=1 then
		旋转气缸:=1;
		Y轴绝对运动位置设定:=-188;
		Y轴绝对运动速度设定:=50;
		Y轴绝对运动启动:=1;
		Z轴绝对运动启动:=0;
		第一个:=1;
END_IF
if Z轴实时位置=135 and X轴实时位置=12 and 取得是10=1 and x2=1 then
		旋转气缸:=1;
		Y轴绝对运动位置设定:=-188;
		Y轴绝对运动速度设定:=50;
		Y轴绝对运动启动:=1;
		Z轴绝对运动启动:=0;
		第一个:=1;
END_IF
if X轴实时位置=572 and 取得是11=1 and x2=1 then
		旋转气缸:=1;
		Y轴绝对运动位置设定:=-188;
		Y轴绝对运动速度设定:=50;
		Y轴绝对运动启动:=1;
		y3 :=1;
		Z轴绝对运动启动:=0;
END_IF

if X轴实时位置=432 and 取得是12=1 and x2=1 then
		旋转气缸:=1;
		Y轴绝对运动位置设定:=-188;
		Y轴绝对运动速度设定:=50;
		Y轴绝对运动启动:=1;
		y3 :=1;
END_IF

if X轴实时位置=292 and 取得是13=1 and x2=1 then
		旋转气缸:=1;
		Y轴绝对运动位置设定:=-188;
		Y轴绝对运动速度设定:=50;
		Y轴绝对运动启动:=1;
		y3 :=1;
END_IF

if X轴实时位置=152 and 取得是14=1 and x2=1 then
		旋转气缸:=1;
		Y轴绝对运动位置设定:=-188;
		Y轴绝对运动速度设定:=50;
		Y轴绝对运动启动:=1;
		y3 :=1;
END_IF
if X轴实时位置=12 and 取得是15=1 and x2=1 then
		旋转气缸:=1;
		Y轴绝对运动位置设定:=-188;
		Y轴绝对运动速度设定:=50;
		Y轴绝对运动启动:=1;
		y3 :=1;
END_IF
if Y轴实时位置=-188 and Z轴实时位置<0 and x2=1 then
	X轴绝对运动启动:=0;
	Z轴绝对运动启动:=0;
	Y轴绝对运动启动:=0;
	夹爪气缸:=1;

	Z轴绝对运动位置设定:=-5;
	Y轴绝对运动位置设定:=40;
	Z轴绝对运动速度设定:=40;
	Y轴绝对运动速度设定:=50;
	X轴绝对运动位置设定:=303;

	夹爪完了:=1;
END_IF
if Y轴实时位置=-188 and Z轴实时位置=280 and x2=1 then
	X轴绝对运动启动:=0;
	Z轴绝对运动启动:=0;
	Y轴绝对运动启动:=0;
	夹爪气缸:=1;

	Z轴绝对运动位置设定:=285;
	Y轴绝对运动位置设定:=40;
	Z轴绝对运动速度设定:=40;
	Y轴绝对运动速度设定:=50;
	X轴绝对运动位置设定:=303;

	夹爪完了:=1;
END_IF
if Y轴实时位置=-188 and Z轴实时位置=135 and x2=1 then
	X轴绝对运动启动:=0;
	Z轴绝对运动启动:=0;
	Y轴绝对运动启动:=0;
	夹爪气缸:=1;

	Z轴绝对运动位置设定:=140;
	Y轴绝对运动位置设定:=40;
	Z轴绝对运动速度设定:=40;
	Y轴绝对运动速度设定:=50;
	X轴绝对运动位置设定:=303;

	夹爪完了:=1;
END_IF
TONR(IN := 夹爪完了,PT := 1000,Q => 开始带走);
TONR(IN := 夹爪完了,PT := 1200,Q => 开始带走2);
IF 开始带走=1 and 回收作业启动=0 and x2=1 THEN
	Z轴绝对运动启动:=1;

	运动状态:=0;
	取料终:=1;
END_IF;
if 开始带走2=1 and 回收作业启动=0 and x2=1 THEN
	Y轴绝对运动启动:=1;
END_if
IF 取料终=1 and Y轴实时位置>35 and x2=1 THEN
	旋转气缸:=0;
	X轴绝对运动启动:=1;
	放到顶上了:=1;
	Z轴绝对运动启动:=0;
	Y轴绝对运动启动:=0;

END_IF;

IF 放到顶上了=1 and X轴实时位置=303 and x2=1 THEN
	Z轴绝对运动位置设定:=0;
	Z轴绝对运动启动:=1;
	Y轴绝对运动启动:=1;
	X轴绝对运动启动:=1;

	放完了:=1;
END_IF;
TONR(IN := 放完了,PT := 200,Q => 真放完了);
IF 真放完了=1 and x2=1 THEN
	Z轴绝对运动启动:=0;
END_IF;
IF 放完了=1 and Z轴实时位置=0 and x2=1 THEN

	夹爪气缸:=0;
	最后放完了:=1;
	绝对放完了:=1;

END_IF;
TONR(IN := 最后放完了,PT := 200,Q => 最后放完了延时);

IF 最后放完了延时=1 and x2=1 THEN
	Z轴绝对运动位置设定:=40;
	Z轴绝对运动启动:=1;
	绝对放完了:=1;
END_IF;
IF Z轴实时位置>39 and 绝对放完了=1 and x2=1 THEN
	x回原点:=1;

	z回原点:=1;
	旋转气缸:=0;
	y轴动作延时:=1;
	方形物料推料气缸:=1;
END_IF;
IF 一号传感器=1 and x2=1 THEN
	六轴机器人启动:=0;
END_IF;
if 二号传感器=1 and x2=1 THEN
	六轴机器人动作预备:=1;
END_IF
TONR(IN := y轴动作延时,PT := 10000,Q => y回原);
TONR(IN := 六轴机器人动作预备,PT := 7000,Q => 六轴机器人动作);
IF y回原=1 and x2=1 THEN
	y回原点:=1;
	X轴绝对运动启动:=0;
	Y轴绝对运动启动:=0;
	Z轴绝对运动启动:=0;
END_IF;
IF 六轴机器人动作=1 and 放完了=1 and x2=1 THEN
	六轴机器人启动:=1;
	六轴机器人动作预备:=0;

END_IF;
if 六轴作业完成=1 and 二号物料完工=0 and 绝对放完了=1 and x2=1 THEN
	二号物料完工:=1;
	方形物料推料气缸:=0;
	END_IF
TONR(IN := 二号物料完工,PT := 21000,Q => 三号物料完工);
TONR(IN := 二号物料完工,PT := 3500,Q => 第三个第二);
TONR(IN := 二号物料完工,PT := 42000,Q => 四号物料完工);
IF 第三个第二=1 and x2=1 THEN
	方形物料推料气缸:=1;
END_IF;
IF 三号物料完工=1 and x2=1 THEN

	方形物料推料气缸:=0;
END_IF;
IF 四号物料完工=1 and x2=1 THEN
	圆形物料推料气缸:=1;
END_IF;
if 四号物料完工=1 and 六轴作业完成=1 and 四号完了=0 and x2=1 then
	回收作业启动:=1;
	圆形物料推料气缸:=0;
	夹爪气缸:=0;
	四号完了:=1;
	y2:=1;
END_IF
IF 回收作业启动=1 and 确保一次启动=0 and x2=1 THEN
	X轴绝对运动位置设定:=303;
	Y轴绝对运动位置设定:=40;
	Z轴绝对运动位置设定:=20;

	回收延时:=1;
	确保一次启动:=1;
END_IF;
TONR(IN := 回收延时,PT := 2000,Q => 回收启动);
IF (X4=1 or 回收启动=1) and x2=1 and 启动只执行一次=0 THEN
	X轴绝对运动启动:=1;
	Y轴绝对运动启动:=1;
	Z轴绝对运动启动:=1;
	回收启动:=0;
	启动只执行一次:=1;
END_IF;

IF 回收作业启动=1 and X轴实时位置=303 and Y轴实时位置=40 and x2=1 THEN
	y0:=1;
	Z轴绝对运动启动:=1;

END_IF;

IF 回收作业启动=1 and x轴回收只执行一次=0 and Y轴实时位置=40 and x2=1 THEN
	Z轴绝对运动启动:=0;
	Z轴绝对运动位置设定:=0;
	x轴回收只执行一次:=1;
	y1:=1;
END_IF;

(* ---- d517.st ---- *)
if M8000=1 and 初始启动一次=0 and x2=1 and 流程=0 THEN
	Z轴绝对运动启动:=0;
	X轴绝对运动启动:=0;
	Y轴绝对运动启动:=0;
	x回原点:=0;
	y回原点:=0;
	z回原点:=0;
	X轴绝对运动速度设定:=50;
	Z轴绝对运动速度设定:=50;

	d1301:=0;
	三轴启动:=0;

	初始启动一次:=1;

END_IF
TONR(IN := 圆形开始,PT := 3000,Q => 圆形延时);
IF x2=0 AND 圆形物料推料气缸=1 THEN
	圆形开始:=1;
END_IF;
IF x2=0 and 圆形延时=1 THEN
	圆形物料推料气缸:=0;

END_IF;
IF (三轴启动=1 or x0=1)  and x2=1 and 流程=0  THEN
	传送带速度:=50;
	传送带位置:=20000;

	切换吸盘:=1;

	X轴绝对运动速度设定:=50;
	Z轴绝对运动速度设定:=50;
	CASE 第一个运行 OF
		1:取出物料盒1:=1;
		2:取出物料盒2:=1;
		3:取出物料盒3:=1;
		4:取出物料盒4:=1;
		5:取出物料盒5:=1;
		6:取出物料盒6:=1;
		7:取出物料盒7:=1;
		8:取出物料盒8:=1;
		9:取出物料盒9:=1;
		10:取出物料盒10:=1;
		11:取出物料盒11:=1;
		12:取出物料盒12:=1;
		13:取出物料盒13:=1;
		14:取出物料盒14:=1;
		15:取出物料盒15:=1;

	Z轴绝对运动启动:=0;
	X轴绝对运动启动:=0;
	END_CASE;
END_IF;
if 取出物料盒1=1 and 取出物料盒只执行一次确保=0 and x2=1 and 流程=0  THEN
	取出1:=1;
	X轴绝对运动位置设定 := 572;
    Z轴绝对运动位置设定 := 280;
	Z轴绝对运动启动:=1;
	取得是1:=1;
	取出物料盒只执行一次确保:=1;
END_IF
if 取出物料盒2=1 and 取出物料盒只执行一次确保=0 and x2=1 and 流程=0  THEN
	取出1:=1;
	X轴绝对运动位置设定 := 432;
    Z轴绝对运动位置设定 := 280;
	Z轴绝对运动启动:=1;
	取得是2:=1;
	取出物料盒只执行一次确保:=1;
END_IF
if  取出物料盒3=1 and 取出物料盒只执行一次确保=0 and x2=1 and 流程=0   THEN
	取出1:=1;
	X轴绝对运动位置设定 := 292;
    Z轴绝对运动位置设定 := 280;
	Z轴绝对运动启动:=1;
	取得是3:=1;
	取出物料盒只执行一次确保:=1;
END_IF
if 取出物料盒4=1 and 取出物料盒只执行一次确保=0 and x2=1 and 流程=0  THEN
	取出1:=1;
	X轴绝对运动位置设定 := 152;
    Z轴绝对运动位置设定 := 280;
	Z轴绝对运动启动:=1;
	取得是4:=1;
	取出物料盒只执行一次确保:=1;
END_IF
if  取出物料盒5=1 and 取出物料盒只执行一次确保=0 and x2=1 and 流程=0  THEN
	取出1:=1;
	X轴绝对运动位置设定 := 12;
    Z轴绝对运动位置设定 := 280;
	Z轴绝对运动启动:=1;
	取得是5:=1;
	取出物料盒只执行一次确保:=1;
END_IF
if 取出物料盒6=1 and 取出物料盒只执行一次确保=0 and x2=1 and 流程=0  THEN
	取出1:=1;
	X轴绝对运动位置设定 := 572;
    Z轴绝对运动位置设定 := 135;
	Z轴绝对运动启动:=1;
	取得是6:=1;
	取出物料盒只执行一次确保:=1;

END_IF
if 取出物料盒7=1 and 取出物料盒只执行一次确保=0  and x2=1 and 流程=0  THEN
	取出1:=1;
	X轴绝对运动位置设定 := 432;
    Z轴绝对运动位置设定 := 135;
	Z轴绝对运动启动:=1;
	取得是7:=1;
	取出物料盒只执行一次确保:=1;
END_IF
if  取出物料盒8=1 and 取出物料盒只执行一次确保=0  and x2=1 and 流程=0  THEN
	取出1:=1;
	X轴绝对运动位置设定 := 292;
    Z轴绝对运动位置设定 := 135;
	Z轴绝对运动启动:=1;
	取得是8:=1;
	取出物料盒只执行一次确保:=1;
END_IF
if 取出物料盒9=1 and 取出物料盒只执行一次确保=0 and x2=1 and 流程=0  THEN
	取出1:=1;
	X轴绝对运动位置设定 := 152;
    Z轴绝对运动位置设定 := 135;
	Z轴绝对运动启动:=1;
	取得是9:=1;
	取出物料盒只执行一次确保:=1;
END_IF
if  取出物料盒10=1 and 取出物料盒只执行一次确保=0 and x2=1  and 流程=0 THEN
	取出1:=1;
	X轴绝对运动位置设定 := 12;
    Z轴绝对运动位置设定 := 135;
	Z轴绝对运动启动:=1;
	取得是10:=1;
	取出物料盒只执行一次确保:=1;
END_IF
if 取出物料盒11=1 and 取出物料盒只执行一次确保=0 and x2=1 and 流程=0  THEN
	取出1:=1;
	X轴绝对运动位置设定 := 572;
    Z轴绝对运动位置设定 := -10;
	Z轴绝对运动启动:=1;
	取得是11:=1;
	取出物料盒只执行一次确保:=1;
END_IF
if 取出物料盒12=1 and 取出物料盒只执行一次确保=0 and x2=1 and 流程=0  THEN
	取出1:=1;
	X轴绝对运动位置设定 := 432;
    Z轴绝对运动位置设定 := -10;
	Z轴绝对运动启动:=1;
	取得是12:=1;
	取出物料盒只执行一次确保:=1;
END_IF
if  取出物料盒13=1 and 取出物料盒只执行一次确保=0  and x2=1 and 流程=0  THEN
	取出1:=1;
	X轴绝对运动位置设定 := 292;
    Z轴绝对运动位置设定 := -10;
	Z轴绝对运动启动:=1;
	取得是13:=1;
	取出物料盒只执行一次确保:=1;
END_IF
if 取出物料盒14=1 and 取出物料盒只执行一次确保=0 and x2=1 and 流程=0  THEN
	取出1:=1;
	X轴绝对运动位置设定 := 152;
    Z轴绝对运动位置设定 := -10;
	Z轴绝对运动启动:=1;
	取得是14:=1;
	取出物料盒只执行一次确保:=1;
END_IF
if  取出物料盒15=1 and 取出物料盒只执行一次确保=0  and x2=1 and 流程=0  THEN
	取出1:=1;
	X轴绝对运动位置设定 := 12;
    Z轴绝对运动位置设定 := -10;
	Z轴绝对运动启动:=1;
	取得是15:=1;
	取出物料盒只执行一次确保:=1;
END_IF
	IF Z轴实时位置>20 and 取得是1=1 and 确保x轴只动一次=0 and 回收作业启动=0 and x2=1 and 流程=0  THEN
		确保x轴只动一次:=1;
		X轴绝对运动启动:=1;
	END_IF;
	IF Z轴实时位置>20 and 取得是2=1 and 确保x轴只动一次=0 and 回收作业启动=0 and x2=1  and 流程=0  THEN
		确保x轴只动一次:=1;
		X轴绝对运动启动:=1;
		传送带启动:=1;
	END_IF;

	IF Z轴实时位置>20 and 取得是3=1 and 确保x轴只动一次=0 and 回收作业启动=0 and x2=1 and 流程=0   THEN
		确保x轴只动一次:=1;
		X轴绝对运动启动:=1;
	END_IF;

	IF Z轴实时位置>20 and 取得是4=1 and 确保x轴只动一次=0 and 回收作业启动=0  and x2=1 and 流程=0  THEN
		确保x轴只动一次:=1;
		X轴绝对运动启动:=1;
	END_IF;

	IF Z轴实时位置>20 and 取得是5=1 and 确保x轴只动一次=0 and 回收作业启动=0  and x2=1 and 流程=0  THEN
		确保x轴只动一次:=1;
		X轴绝对运动启动:=1;
	END_IF;
	IF Z轴实时位置>20 and 取得是6=1 and 确保x轴只动一次=0 and 回收作业启动=0 and x2=1 and 流程=0  THEN
		确保x轴只动一次:=1;

		X轴绝对运动启动:=1;
		传送带启动:=1;
	END_IF;
	IF Z轴实时位置>20 and 取得是7=1 and 确保x轴只动一次=0 and 回收作业启动=0 and x2=1 and 流程=0   THEN
		确保x轴只动一次:=1;
		X轴绝对运动启动:=1;
		传送带启动:=1;
	END_IF;

	IF Z轴实时位置>20 and 取得是8=1 and 确保x轴只动一次=0 and 回收作业启动=0 and x2=1  and 流程=0  THEN
		确保x轴只动一次:=1;
		X轴绝对运动启动:=1;
	END_IF;

	IF Z轴实时位置>20 and 取得是9=1 and 确保x轴只动一次=0 and 回收作业启动=0 and x2=1 and 流程=0   THEN
		确保x轴只动一次:=1;
		X轴绝对运动启动:=1;
	END_IF;

	IF Z轴实时位置>20 and 取得是10=1 and 确保x轴只动一次=0 and 回收作业启动=0 and x2=1  and 流程=0  THEN
		确保x轴只动一次:=1;
		X轴绝对运动启动:=1;
	END_IF;
	IF Z轴实时位置<-2 and 取得是11=1 and 确保x轴只动一次=0 and 回收作业启动=0 and x2=1 and 流程=0  THEN
		确保x轴只动一次:=1;
		X轴绝对运动启动:=1;
	END_IF;
	IF Z轴实时位置<-2 and 取得是12=1 and 确保x轴只动一次=0 and 回收作业启动=0  and x2=1 and 流程=0  THEN
		确保x轴只动一次:=1;
		X轴绝对运动启动:=1;
		传送带启动:=1;
	END_IF;

	IF Z轴实时位置<-2 and 取得是13=1 and 确保x轴只动一次=0  and 回收作业启动=0 and x2=1 and 流程=0  THEN
		确保x轴只动一次:=1;
		X轴绝对运动启动:=1;
	END_IF;

	IF Z轴实时位置<-2 and 取得是14=1 and 确保x轴只动一次=0  and 回收作业启动=0 and x2=1 and 流程=0  THEN
		确保x轴只动一次:=1;
		X轴绝对运动启动:=1;
	END_IF;

	IF Z轴实时位置<-2 and 取得是15=1 and 确保x轴只动一次=0 and 回收作业启动=0 and x2=1 and 流程=0  THEN
		确保x轴只动一次:=1;
		X轴绝对运动启动:=1;
	END_IF;
IF Z轴实时位置>30 and 第一个=0 and 回收作业启动=0 and x2=1 and 流程=0  THEN

	一号物料完工:=1;
	END_IF
if Z轴实时位置=280 and X轴实时位置=572 and 取得是1=1 and x2=1 and 流程=0  then
		旋转气缸:=1;
		Y轴绝对运动位置设定:=-188;
		Y轴绝对运动速度设定:=50;
		Y轴绝对运动启动:=1;
		Z轴绝对运动启动:=0;
		第一个:=1;
END_IF

if Z轴实时位置=280 and X轴实时位置=432 and 取得是2=1 and x2=1 and 流程=0  then
		旋转气缸:=1;
		Y轴绝对运动位置设定:=-188;
		Y轴绝对运动速度设定:=50;
		Y轴绝对运动启动:=1;
		Z轴绝对运动启动:=0;
		第一个:=1;
END_IF

if Z轴实时位置=280 and X轴实时位置=292 and 取得是3=1 and x2=1 and 流程=0  then
		旋转气缸:=1;
		Y轴绝对运动位置设定:=-188;
		Y轴绝对运动速度设定:=50;
		Y轴绝对运动启动:=1;
		Z轴绝对运动启动:=0;
		第一个:=1;
END_IF

if Z轴实时位置=280 and X轴实时位置=152 and 取得是4=1 and x2=1 and 流程=0  then
		旋转气缸:=1;
		Y轴绝对运动位置设定:=-188;
		Y轴绝对运动速度设定:=50;
		Y轴绝对运动启动:=1;
		Z轴绝对运动启动:=0;
		第一个:=1;
END_IF
if Z轴实时位置=280 and X轴实时位置=12 and 取得是5=1 and x2=1 and 流程=0  then
		旋转气缸:=1;
		Y轴绝对运动位置设定:=-188;
		Y轴绝对运动速度设定:=50;
		Y轴绝对运动启动:=1;
		Z轴绝对运动启动:=0;
		第一个:=1;
END_IF
if Z轴实时位置=135 and X轴实时位置=572 and 取得是6=1 and x2=1 and 流程=0  then
		旋转气缸:=1;
		Y轴绝对运动位置设定:=-188;
		Y轴绝对运动速度设定:=50;
		Y轴绝对运动启动:=1;

		Z轴绝对运动启动:=0;
		第一个:=1;
END_IF

if Z轴实时位置=135 and X轴实时位置=432 and 取得是7=1 and x2=1 and 流程=0  then
		旋转气缸:=1;
		Y轴绝对运动位置设定:=-188;
		Y轴绝对运动速度设定:=50;
		Y轴绝对运动启动:=1;
		Z轴绝对运动启动:=0;
		第一个:=1;
END_IF

if Z轴实时位置=135 and X轴实时位置=292 and 取得是8=1 and x2=1 and 流程=0  then
		旋转气缸:=1;
		Y轴绝对运动位置设定:=-188;
		Y轴绝对运动启动:=1;
		Z轴绝对运动启动:=0;
		第一个:=1;
END_IF

if Z轴实时位置=135 and X轴实时位置=152 and 取得是9=1 and x2=1  and 流程=0 then
		旋转气缸:=1;
		Y轴绝对运动位置设定:=-188;
		Y轴绝对运动速度设定:=50;
		Y轴绝对运动启动:=1;
		Z轴绝对运动启动:=0;
		第一个:=1;
END_IF
if Z轴实时位置=135 and X轴实时位置=12 and 取得是10=1 and x2=1 and 流程=0  then
		旋转气缸:=1;
		Y轴绝对运动位置设定:=-188;
		Y轴绝对运动速度设定:=50;
		Y轴绝对运动启动:=1;
		Z轴绝对运动启动:=0;
		第一个:=1;
END_IF
if X轴实时位置=572 and 取得是11=1 and x2=1 and 流程=0  then
		旋转气缸:=1;
		Y轴绝对运动位置设定:=-188;
		Y轴绝对运动速度设定:=50;
		Y轴绝对运动启动:=1;
		y3 :=1;
		Z轴绝对运动启动:=0;
END_IF

if X轴实时位置=432 and 取得是12=1 and x2=1 and 流程=0  then
		旋转气缸:=1;
		Y轴绝对运动位置设定:=-188;
		Y轴绝对运动速度设定:=50;
		Y轴绝对运动启动:=1;
		y3 :=1;
END_IF

if X轴实时位置=292 and 取得是13=1 and x2=1 and 流程=0  then
		旋转气缸:=1;
		Y轴绝对运动位置设定:=-188;
		Y轴绝对运动速度设定:=50;
		Y轴绝对运动启动:=1;
		y3 :=1;
END_IF

if X轴实时位置=152 and 取得是14=1 and x2=1 and 流程=0  then
		旋转气缸:=1;
		Y轴绝对运动位置设定:=-188;
		Y轴绝对运动速度设定:=50;
		Y轴绝对运动启动:=1;
		y3 :=1;
END_IF
if X轴实时位置=12 and 取得是15=1 and x2=1 and 流程=0  then
		旋转气缸:=1;
		Y轴绝对运动位置设定:=-188;
		Y轴绝对运动速度设定:=50;
		Y轴绝对运动启动:=1;
		y3 :=1;
END_IF
if Y轴实时位置=-188 and Z轴实时位置<0 and x2=1 and 流程=0  then
	X轴绝对运动启动:=0;
	Z轴绝对运动启动:=0;
	Y轴绝对运动启动:=0;
	夹爪气缸:=1;

	Z轴绝对运动位置设定:=-5;
	Y轴绝对运动位置设定:=40;
	Z轴绝对运动速度设定:=40;
	Y轴绝对运动速度设定:=50;
	X轴绝对运动位置设定:=303;

	夹爪完了:=1;
END_IF
if Y轴实时位置=-188 and Z轴实时位置=280 and x2=1 and 流程=0  then
	X轴绝对运动启动:=0;
	Z轴绝对运动启动:=0;
	Y轴绝对运动启动:=0;
	夹爪气缸:=1;

	Z轴绝对运动位置设定:=285;
	Y轴绝对运动位置设定:=40;
	Z轴绝对运动速度设定:=40;
	Y轴绝对运动速度设定:=50;
	X轴绝对运动位置设定:=303;

	夹爪完了:=1;
END_IF
if Y轴实时位置=-188 and Z轴实时位置=135 and x2=1 and 流程=0  then
	X轴绝对运动启动:=0;
	Z轴绝对运动启动:=0;
	Y轴绝对运动启动:=0;
	夹爪气缸:=1;

	Z轴绝对运动位置设定:=140;
	Y轴绝对运动位置设定:=40;
	Z轴绝对运动速度设定:=40;
	Y轴绝对运动速度设定:=50;
	X轴绝对运动位置设定:=303;

	夹爪完了:=1;
END_IF
TONR(IN := 夹爪完了,PT := 1000,Q => 开始带走);
TONR(IN := 夹爪完了,PT := 1200,Q => 开始带走2);
IF 开始带走=1 and 回收作业启动=0 and x2=1 and 流程=0  THEN
	Z轴绝对运动启动:=1;

	运动状态:=0;
	取料终:=1;
END_IF;
if 开始带走2=1 and 回收作业启动=0 and x2=1 and 流程=0  THEN
	Y轴绝对运动启动:=1;
END_if
IF 取料终=1 and Y轴实时位置>35 and x2=1 and 流程=0  THEN
	旋转气缸:=0;
	X轴绝对运动启动:=1;
	放到顶上了:=1;
	Z轴绝对运动启动:=0;
	Y轴绝对运动启动:=0;

END_IF;

IF 放到顶上了=1 and X轴实时位置=303 and x2=1 and 流程=0  THEN
	Z轴绝对运动位置设定:=0;
	Z轴绝对运动启动:=1;
	Y轴绝对运动启动:=1;
	X轴绝对运动启动:=1;

	放完了:=1;
END_IF;
TONR(IN := 放完了,PT := 200,Q => 真放完了);
IF 真放完了=1 and x2=1 and 流程=0  THEN
	Z轴绝对运动启动:=0;
END_IF;
IF 放完了=1 and Z轴实时位置=0 and x2=1 and 流程=0  THEN

	夹爪气缸:=0;
	最后放完了:=1;
	绝对放完了:=1;

END_IF;
TONR(IN := 最后放完了,PT := 200,Q => 最后放完了延时);

IF 最后放完了延时=1 and x2=1 and 流程=0  THEN
	Z轴绝对运动位置设定:=40;
	Z轴绝对运动启动:=1;
	绝对放完了:=1;
END_IF;
IF Z轴实时位置>39 and 绝对放完了=1 and x2=1 and 流程=0  THEN
	x回原点:=1;

	z回原点:=1;
	旋转气缸:=0;
	y轴动作延时:=1;

END_IF;
IF y回原=1 and x2=1 and 流程=0  THEN
	y回原点:=1;
	X轴绝对运动启动:=0;
	Y轴绝对运动启动:=0;
	Z轴绝对运动启动:=0;
END_IF;
//六轴机器人程序区开始

IF 一号传感器=1 and x2=1 and 流程=0  THEN
	六轴机器人启动:=0;
END_IF;
if 二号传感器=1 and x2=1 and 流程=0  THEN
	六轴机器人动作预备:=1;
END_IF
TONR(IN := y轴动作延时,PT := 10000,Q => y回原);
TONR(IN := 六轴机器人动作预备,PT := 8000,Q => 六轴机器人动作);

IF 六轴机器人动作=1 and 放完了=1 and x2=1  and 流程=0 THEN
	六轴机器人启动:=1;
	六轴机器人动作预备:=0;

END_IF;
//六轴机器人程序区结束
//落料程序区开始
TONR(IN := 落下准备,PT := 7000,Q => 落下延时);
	TONR(IN := 落下准备2,PT := 6500,Q => 落下延时2);
	TONR(IN := 落下准备3,PT := 7000,Q => 落下延时3);
	TONR(IN := 落下准备4,PT := 6500,Q => 落下延时4);
	TONR(IN := 落下准备4,PT := 33500,Q =>落料完成);
if (三轴启动=1 or x0=1) and 第一个准备=0 and 流程=0  THEN
	圆形物料推料气缸:=1;
	第一个准备:=1;
	落下准备:=1;
END_IF
IF 落下延时=1 and 落下只执行一次1=0 and 流程=0  THEN
	圆形物料推料气缸:=0;
	第一个落下:=1;
	落下只执行一次1:=1;
END_IF;
IF 第一个落下=1 and 六轴作业完成=1 and 第二个准备=0 and 放完了=1 and 流程=0  THEN
	方形物料推料气缸:=1;
	第二个准备:=1;
	落下准备2:=1;
END_IF;
	IF 落下延时2=1 and 落下只执行一次2=0 THEN
	方形物料推料气缸:=0;
	第二个落下:=1;
	落下只执行一次2:=1;
END_IF;
IF 第二个落下=1 and 六轴作业完成=1 and 第三个准备=0 and 流程=0  THEN
	方形物料推料气缸:=1;
	第三个准备:=1;
	落下准备3:=1;
END_IF;
	IF 落下延时3=1 and 落下只执行一次3=0 and 流程=0  THEN
	方形物料推料气缸:=0;
	第三个落下:=1;
	落下只执行一次3:=1;
END_IF;
	IF 第三个落下=1 and 六轴作业完成=1 and 第四个准备=0 and 流程=0  THEN
	圆形物料推料气缸:=1;
	第四个准备:=1;
	落下准备4:=1;
END_IF;
	IF 落下延时4=1 and 落下只执行一次4=0 and 流程=0  THEN
	圆形物料推料气缸:=0;
	第四个落下:=1;
	落下只执行一次4:=1;
END_IF;
//落料程序区结束
IF x5=1 THEN
		流程:=3;
END_IF;

IF 落料完成=1 and 确保一次启动=0 and x2=1 THEN
	流程:=3;
	X轴绝对运动位置设定:=303;
	Y轴绝对运动位置设定:=40;

	Z轴绝对运动位置设定:=10;
	Y轴绝对运动启动:=1;
	Z轴绝对运动启动:=1;
	取出物料盒只执行一次确保:=1;
	确保一次启动:=1;
END_IF;

if 流程=3 and x2=1 and Y轴实时位置>20 and Y轴实时位置<30 THEN
	X轴绝对运动启动:=1;
	Y轴绝对运动启动:=0;
	Z轴绝对运动启动:=0;
	Z轴绝对运动位置设定:=0;
	END_IF
if 流程=3 and x2=1 and X轴实时位置=303 and Z轴实时位置>9.9 THEN
	X轴绝对运动启动:=0;
	Z轴绝对运动启动:=1;
	END_IF
if 流程=3 and x2=1 and X轴实时位置=303 and Z轴实时位置=0 THEN
	夹爪气缸:=1;
	Z轴绝对运动启动:=0;
	Z轴绝对运动位置设定:=30;
	抓住:=1;
	END_IF
TONR(IN := 抓住,PT := 2000,Q => 抓住延时);
if 流程=3 and x2=1 and 抓住延时=1 and Z轴实时位置=0 THEN
	Z轴绝对运动启动:=1;
	END_IF

if 流程=3 and x2=1 and 抓住延时=1 and Z轴实时位置>29.9 and 取得是6=1 and Z轴实时位置<35 THEN
	旋转气缸:=1;
	X轴绝对运动位置设定 := 572;
    Z轴绝对运动位置设定 := 150;
	Z轴绝对运动启动:=0;
	X轴绝对运动启动:=0;
	放过去:=1;
	END_IF
if 流程=3 and x2=1 and 抓住延时=1 and X轴实时位置=572 and Z轴实时位置=150 and 取得是6=1 THEN
	Y轴绝对运动位置设定:=-188;
	Z轴绝对运动启动:=0;
	X轴绝对运动启动:=0;
	Y轴绝对运动启动:=1;
	END_IF
TONR(IN := 放过去,PT := 1000,Q => 放过去延时);
if 流程=3 and x2=1 and 抓住延时=1 and X轴实时位置=303 and 放过去延时=1 THEN
	X轴绝对运动启动:=1;
	Z轴绝对运动启动:=1;
	END_IF
if 流程=3 and x2=1 and 抓住延时=1 and 放过去延时=1 and Y轴实时位置=-188 and Z轴实时位置=150 THEN
	Z轴绝对运动位置设定:=135;
	Z轴绝对运动启动:=0;
	放料:=1;
	X轴绝对运动启动:=0;
	Y轴绝对运动启动:=0;
	Y轴绝对运动位置设定:=20;
	END_IF
TONR(IN := 放料,PT := 1000,Q => 放料延时);
if 流程=3 and x2=1 and 抓住延时=1 and Y轴实时位置=-188 and Z轴实时位置=150 and 放料延时=1 THEN
	Z轴绝对运动启动:=1;
END_IF
if 流程=3 and x2=1 and 抓住延时=1 and Y轴实时位置=-188 and Z轴实时位置=135 and 放料延时=1 THEN
	夹爪气缸:=0;
	Y轴绝对运动启动:=1;
		d1301:=0;
END_IF
if 流程=3 and x2=1 and 抓住延时=1 and Y轴实时位置=20 AND 放料延时=1 THEN
	流程:=0;
	Y轴绝对运动启动:=0;
	Z轴绝对运动启动:=0;
	回收作业启动:=0;
	开始吧:=1;
	取出物料盒只执行一次确保:=0;
	确保x轴只动一次:=0;
	CASE 第二个运行 OF
		1:取出物料盒1:=1;
		2:取出物料盒2:=1;
		3:取出物料盒3:=1;
		4:取出物料盒4:=1;
		5:取出物料盒5:=1;
		6:取出物料盒6:=1;
		7:取出物料盒7:=1;
		8:取出物料盒8:=1;
		9:取出物料盒9:=1;
		10:取出物料盒10:=1;
		11:取出物料盒11:=1;
		12:取出物料盒12:=1;
		13:取出物料盒13:=1;
		14:取出物料盒14:=1;
		15:取出物料盒15:=1;
	X轴绝对运动启动:=0;
	END_CASE;
END_IF

(*IF 流程=5 and 开始吧=1 AND 第二个运行=1 THEN
	X轴绝对运动位置设定 := 572;
    Z轴绝对运动位置设定 := 280;

	开始吧:=0;
	y0:=1;
	取料2:=1;
END_IF;
TONR(IN := 取料2,PT := 500,Q => 取料2延时);
IF 流程=5 and 取料2延时=1 AND 取料2自锁=0 THEN

	Z轴绝对运动启动:=1;
	X轴绝对运动启动:=1;
		取料2自锁:=1;
	y1:=1;
	END_IF

IF 流程=5 and X轴实时位置=572 and Z轴实时位置=280 THEN
	X轴绝对运动启动:=1;
	Y轴绝对运动位置设定:=-188;
	Y轴绝对运动启动:=1;

END_IF;*)
(*if 第二个运行=1 and 取出物料盒只执行一次确保=0 and x2=1 and 流程=5  THEN

	X轴绝对运动位置设定 := 572;
    Z轴绝对运动位置设定 := 280;

	取得是1:=1;
	取出物料盒只执行一次确保:=1;
END_IF
if 第二个运行=2 and 取出物料盒只执行一次确保=0 and x2=1 and 流程=5  THEN

	X轴绝对运动位置设定 := 432;
    Z轴绝对运动位置设定 := 280;

	取得是2:=1;
	取出物料盒只执行一次确保:=1;
END_IF
if  第二个运行=3 and 取出物料盒只执行一次确保=0 and x2=1 and 流程=5   THEN

	X轴绝对运动位置设定 := 292;
    Z轴绝对运动位置设定 := 280;

	取得是3:=1;
	取出物料盒只执行一次确保:=1;
END_IF
if 第二个运行=4 and 取出物料盒只执行一次确保=0 and x2=1 and 流程=5  THEN

	X轴绝对运动位置设定 := 152;
    Z轴绝对运动位置设定 := 280;

	取得是4:=1;
	取出物料盒只执行一次确保:=1;
END_IF
if  第二个运行=5 and 取出物料盒只执行一次确保=0 and x2=1 and 流程=5  THEN

	X轴绝对运动位置设定 := 12;
    Z轴绝对运动位置设定 := 280;

	取得是5:=1;
	取出物料盒只执行一次确保:=1;
END_IF
if 第二个运行=6 and 取出物料盒只执行一次确保=0 and x2=1 and 流程=5  THEN

	X轴绝对运动位置设定 := 572;
    Z轴绝对运动位置设定 := 135;

	取得是6:=1;
	取出物料盒只执行一次确保:=1;

END_IF
if 第二个运行=7 and 取出物料盒只执行一次确保=0  and x2=1 and 流程=5  THEN

	X轴绝对运动位置设定 := 432;
    Z轴绝对运动位置设定 := 135;

	取得是7:=1;
	取出物料盒只执行一次确保:=1;
END_IF
if  第二个运行=8 and 取出物料盒只执行一次确保=0  and x2=1 and 流程=5  THEN

	X轴绝对运动位置设定 := 292;
    Z轴绝对运动位置设定 := 135;

	取得是8:=1;
	取出物料盒只执行一次确保:=1;
END_IF
if 第二个运行=9 and 取出物料盒只执行一次确保=0 and x2=1 and 流程=5  THEN

	X轴绝对运动位置设定 := 152;
    Z轴绝对运动位置设定 := 135;

	取得是9:=1;
	取出物料盒只执行一次确保:=1;
END_IF
if  第二个运行=10 and 取出物料盒只执行一次确保=0 and x2=1  and 流程=5 THEN

	X轴绝对运动位置设定 := 12;
    Z轴绝对运动位置设定 := 135;

	取得是10:=1;
	取出物料盒只执行一次确保:=1;
END_IF
if 第二个运行=11 and 取出物料盒只执行一次确保=0 and x2=1 and 流程=5  THEN

	X轴绝对运动位置设定 := 572;
    Z轴绝对运动位置设定 := -10;

	取得是11:=1;
	取出物料盒只执行一次确保:=1;
END_IF
if 第二个运行=12 and 取出物料盒只执行一次确保=0 and x2=1 and 流程=5  THEN

	X轴绝对运动位置设定 := 432;
    Z轴绝对运动位置设定 := -10;

	取得是12:=1;
	取出物料盒只执行一次确保:=1;
END_IF
if  第二个运行=13 and 取出物料盒只执行一次确保=0  and x2=1 and 流程=5  THEN

	X轴绝对运动位置设定 := 292;
    Z轴绝对运动位置设定 := -10;

	取得是13:=1;
	取出物料盒只执行一次确保:=1;
END_IF
if 第二个运行=14 and 取出物料盒只执行一次确保=0 and x2=1 and 流程=5  THEN

	X轴绝对运动位置设定 := 152;
    Z轴绝对运动位置设定 := -10;

	取得是14:=1;
	取出物料盒只执行一次确保:=1;
END_IF
if  第二个运行=15 and 取出物料盒只执行一次确保=0  and x2=1 and 流程=5  THEN

	X轴绝对运动位置设定 := 12;
    Z轴绝对运动位置设定 := -10;

	取得是15:=1;
	取出物料盒只执行一次确保:=1;
END_IF
IF 流程=5 and x2=1 and Y轴实时位置>0 THEN
	X轴绝对运动启动:=1;
	Z轴绝对运动启动:=1;
END_IF;
*)

(* ---- main.st ---- *)
PROGRAM MainProgram
VAR
    物料位置: INT AT %M1000; (* 中间变量，用于表示物料库位置 *)
    错误_1: BOOL AT %M1001; (* 15个库的报错变量 *)
    错误_2: BOOL AT %M1002;
    错误_3: BOOL AT %M1003;
    错误_4: BOOL AT %M1004;
    错误_5: BOOL AT %M1005;
    错误_6: BOOL AT %M1006;
    错误_7: BOOL AT %M1007;
    错误_8: BOOL AT %M1008;
    错误_9: BOOL AT %M1009;
    错误_10: BOOL AT %M1010;
    错误_11: BOOL AT %M1011;
    错误_12: BOOL AT %M1012;
    错误_13: BOOL AT %M1013;
    错误_14: BOOL AT %M1014;
    错误_15: BOOL AT %M1015;

    X_位置: REAL AT %DB1.DBD0; (* 机器人的X轴位置 *)
    Y_位置: REAL AT %DB1.DBD4; (* 机器人的Y轴位置 *)
    Z_位置: REAL AT %DB1.DBD8; (* 机器人的Z轴位置 *)

    X_速度: REAL AT %DB1.DBD12; (* X轴绝对运动速度 *)
    Y_速度: REAL AT %DB1.DBD16; (* Y轴绝对运动速度 *)
    Z_速度: REAL AT %DB1.DBD20; (* Z轴绝对运动速度 *)

    X_运动启动: BOOL AT %I0.0; (* X轴绝对运动启动 *)
    Y_运动启动: BOOL AT %I0.1; (* Y轴绝对运动启动 *)
    Z_运动启动: BOOL AT %I0.2; (* Z轴绝对运动启动 *)

    X_当前位置: REAL AT %DB1.DBD24; (* 机器人X轴实时位置 *)
    Y_当前位置: REAL AT %DB1.DBD28; (* 机器人Y轴实时位置 *)
    Z_当前位置: REAL AT %DB1.DBD32; (* 机器人Z轴实时位置 *)

END_VAR

(* 在这里编写主逻辑 *)

(* 检查每个库的光电传感器状态 *)
物料位置 := 读取物料位置(); (* 读取物料库位置 *)

CASE 物料位置 OF
    1: 检查物料(1012, 错误_1); (* 检查1号库的光电传感器状态 *)
    2: 检查物料(1013, 错误_2); (* 检查2号库的光电传感器状态 *)
    3: 检查物料(1014, 错误_3); (* 检查3号库的光电传感器状态 *)
    4: 检查物料(1015, 错误_4); (* 检查4号库的光电传感器状态 *)
    5: 检查物料(1016, 错误_5); (* 检查5号库的光电传感器状态 *)
    6: 检查物料(1017, 错误_6); (* 检查6号库的光电传感器状态 *)
    7: 检查物料(1018, 错误_7); (* 检查7号库的光电传感器状态 *)
    8: 检查物料(1019, 错误_8); (* 检查8号库的光电传感器状态 *)
    9: 检查物料(1020, 错误_9); (* 检查9号库的光电传感器状态 *)
    10: 检查物料(1021, 错误_10); (* 检查10号库的光电传感器状态 *)
    11: 检查物料(1022, 错误_11); (* 检查11号库的光电传感器状态 *)
    12: 检查物料(1023, 错误_12); (* 检查12号库的光电传感器状态 *)
    13: 检查物料(1024, 错误_13); (* 检查13号库的光电传感器状态 *)
    14: 检查物料(1025, 错误_14); (* 检查14号库的光电传感器状态 *)
    15: 检查物料(1026, 错误_15); (* 检查15号库的光电传感器状态 *)
ELSE
    (* Do nothing *)
END_CASE

(* 控制机器人到达指定的库位置 *)
IF 物料位置 > 0 THEN
    设置机器人位置(物料位置);
END_IF

(* 读取机器人的实时位置 *)
X_当前位置 := D1028; (* 读取机器人X轴实时位置 *)

(* 以下是各个子函数的定义 *)

FUNCTION 读取物料位置 : INT
    (* 读取物料库位置的逻辑 *)
    (* 返回物料库位置 *)
END_FUNCTION

FUNCTION 检查物料 (传感器地址: INT; var 错误变量: BOOL)
    (* 检查物料库光电传感器状态的逻辑 *)
    (* 如果库中不存在物料，将错误变量置为TRUE *)
    (* 如果库中存在物料，将错误变量置为FALSE *)
    IF 读取传感器(传感器地址) = 0 THEN
        错误变量 := TRUE;
    ELSE
        错误变量 := FALSE;
    END_IF
END_FUNCTION

FUNCTION 设置机器人位置 (位置: INT)
    (* 控制机器人到达指定库位置的逻辑 *)
    (* 将机器人的X/Y/Z轴位置和速度设定为对应的D寄存器值 *)
    (* 启动机器人的X/Y/Z轴绝对运动 *)
END_FUNCTION

FUNCTION 读取传感器 (传感器地址: INT) : INT
    (* 读取光电传感器状态的逻辑 *)
    (* 返回传感器状态，如果有物料则返回1，否则返回0 *)
END_FUNCTION
